Universal Robots PolyScope program: omer1.urp

Program omer1 (installation=default createdIn=3.15.6 lastSavedIn=3.15.6)
Robot Program (runOnlyOnce=true)
  Script file omer1.script
    | def Program():
    |   extruderTcp = p[0.00374, 0.0002, 0.24259, 0, 3.14159, 0]
    |   extruderWeight = 0.8
    |   extruderCog = [0.00374, 0.0002, 0.24259]
    |   Speed000 = 0.2
    |   Zone000 = 0.02
    |   set_tcp(extruderTcp)
    |   set_payload(extruderWeight, extruderCog)
    |   movej([0, -0.7854, 1.1345, -1.9199, -1.5708, -1.5708], a=3.1416, v=0.6283, r=Zone000)
    |   movej([0, -0.7854, 1.1345, -1.9199, -1.5708, -1.5708], a=3.1416, v=0.6283, r=Zone000)
    | end
    | Program()
